SUBAPPLICATION HebenSenken_ILOCK_QDA_PWM_OPC (* 2 Remote-Kommandos (Heben/Senken, je Subscribe+State-Publish, ODER-verknuepft mit IO-Test wie bei ILOCK_SWITCH_2_QXA_OPC) auf 1 ratiometrisches PWM-Signal (Danfoss PVEA: 25%=Senken, 50%=Neutral, 75%=Heben, Lastteiler-korrigiert). ILOCK_SWITCH_PROTECT_AX (Last-Wins mit Schutzzeit) sorgt dafuer, dass Heben und Senken nie gleichzeitig aktiv sind. Generisch fuer jeden PVEA-Aktor mit ratiometrischem 3-Stufen-PWM-Kanal. *)
  (* Standard: 61499-2 *)
  (* Version 1.3, 2026-09-27, Franz Höpfinger, Meisterschulen am Ostbahnhof, Franz: 'HebenSenken_ILOCK_QDA_PWM_OPC sehe ich KEINE Aenderung?' - das eigene Mux/Skalierungs/Ausgabe-Teilnetz (ASSEMBLE_AB_FROM_AX/AB_TO_AUI/values_50_75_25/AR_AUI_MUX_3/AR_R_MUL_Korrektur/AR_R_MUL_PWM13BIT/AR_TO_AD_NUM/DigitalOutput_PWM) war seit der Auslagerung nach MyLib::sys::HebenSenken_QDA_PWM (fuer Bunkerboden_PWM) doppelt vorhanden - jetzt durch eine Instanz von HebenSenken_QDA_PWM ersetzt (HEBEN/SENKEN aus SPLIT_HEBEN_OUT/SPLIT_SENKEN_OUT direkt verdrahtet statt vorher inline), unveraendertes Verhalten, keine Duplizierung mehr. *)
  (* Version 1.2, 2026-09-27, Franz Höpfinger, Meisterschulen am Ostbahnhof, AR_R_MUL_Korrektur/AR_R_MUL_PWM13BIT FACTOR von eingebackenen Rohwerten (REAL#0.715/REAL#81.91) auf benannte Konstanten aus der neuen MyLib::sys::const::PWM_Konstanten umgestellt (PWM_LASTTEILER_KORREKTUR/PWM_13BIT_SKALIERUNG) - unveraendertes Verhalten, nur nicht mehr an mehreren Stellen als Rohwert wiederholt. values_50_75_25 bekommt jetzt explizit FACTOR_75/FACTOR_25 aus derselben GCF (VALUES_50_75_25_FACTOR_75/_25), seit values_50_75_25 v1.2 eigene Parameter statt eingebackener Werte. *)
  (* Version 1.1, 2026-09-20, Franz Höpfinger, Meisterschulen am Ostbahnhof, PWM_POW von intern fest verdrahtetem initval_AR (1.0) auf einen eigenen Socket umgestellt - ein generischer, wiederverwendbarer Typ darf keinen Fixwert fuer eine Groesse verdrahten, die pro Instanz unterschiedlich sein soll (z.B. Aufnahme_Rechts_KVE16_Reserve.SUB braucht ggf. eine andere Verdrahtung als Aufnahme_Links). *)
  (* Version 1.0, 2026-09-08, Franz Höpfinger, Meisterschulen am Ostbahnhof, Ausgelagert aus Heben_Senken_TO_QDA_PWM_OPC (PWM/ILOCK/Mux-Teilnetz, ohne die Freigabe-DO) zur Wiederverwendung. *)
  PACKAGE MyLib::sys;
  IMPORT logiBUS::io::DQ::logiBUS_DO;
  IMPORT logiBUS::io::DQ::logiBUS_DO_S;
  IMPORT MyLib::sys::const::PWM_Konstanten::PWM_LASTTEILER_KORREKTUR;
  IMPORT MyLib::sys::const::PWM_Konstanten::PWM_13BIT_SKALIERUNG;
  IMPORT MyLib::sys::const::PWM_Konstanten::VALUES_50_75_25_FACTOR_75;
  IMPORT MyLib::sys::const::PWM_Konstanten::VALUES_50_75_25_FACTOR_25;
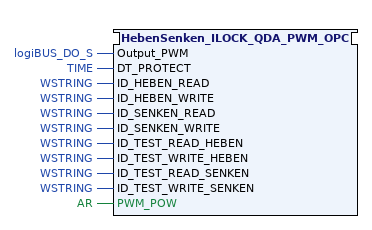
  VAR_INPUT
    Output_PWM : logiBUS::io::DQ::logiBUS_DO_S := logiBUS_DO::Invalid; (* Physischer PWM-Ausgang: 25/50/75% Tastgrad, ratiometrisch *)
    DT_PROTECT : TIME := T#300ms; (* Schutz-Totzeit vor Richtungswechsel *)
    ID_HEBEN_READ : WSTRING; (* Echtes Funktions-Kommando Heben (Subscribe) *)
    ID_HEBEN_WRITE : WSTRING; (* Echte Funktions-Rueckmeldung Heben, HINTER dem ILOCK (Publish) *)
    ID_SENKEN_READ : WSTRING; (* Echtes Funktions-Kommando Senken (Subscribe) *)
    ID_SENKEN_WRITE : WSTRING; (* Echte Funktions-Rueckmeldung Senken, HINTER dem ILOCK (Publish) *)
    ID_TEST_READ_HEBEN : WSTRING; (* Bestehende IO-Test-Subscribe-Adresse Heben (z.B. STG2_Q0x_READ), ODER-verknuepft mit ID_HEBEN_READ vor dem ILOCK *)
    ID_TEST_WRITE_HEBEN : WSTRING; (* Bestehende IO-Test-Publish-Adresse Heben, HINTER dem ILOCK (z.B. STG2_Q0x_WRITE) *)
    ID_TEST_READ_SENKEN : WSTRING; (* Bestehende IO-Test-Subscribe-Adresse Senken, ODER-verknuepft mit ID_SENKEN_READ vor dem ILOCK *)
    ID_TEST_WRITE_SENKEN : WSTRING; (* Bestehende IO-Test-Publish-Adresse Senken, HINTER dem ILOCK *)
  END_VAR
  SOCKETS
    PWM_POW : adapter::types::unidirectional::AR; (* PWM Power 1.0 = Maximale Power, 0.0 = Aus, 0.5 = Halb - durchgereicht an values_50_75_25.PWM_POW *)
  END_SOCKETS
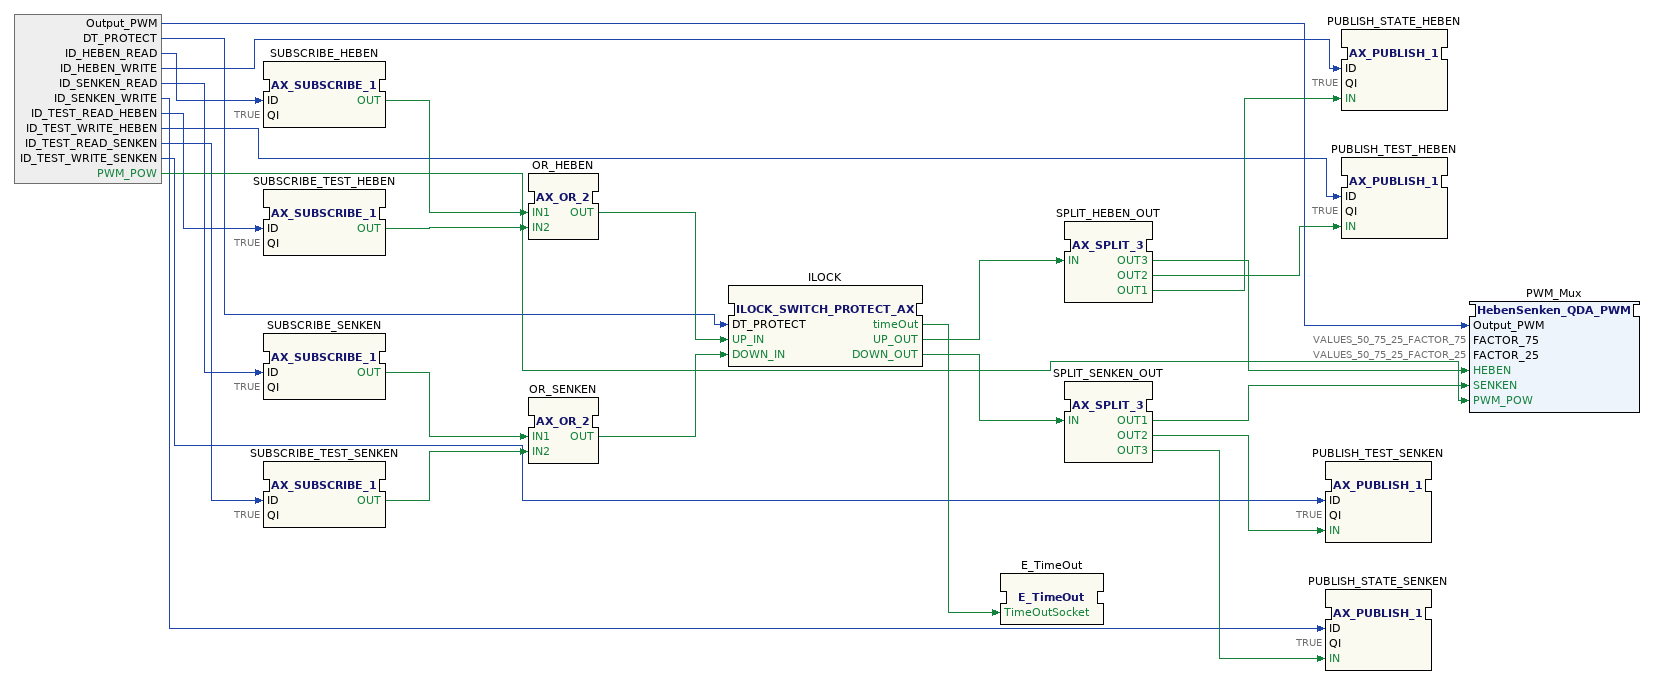
  FBS
    SUBSCRIBE_HEBEN : adapter::net::AX_SUBSCRIBE_1(QI := TRUE);
    SUBSCRIBE_TEST_HEBEN : adapter::net::AX_SUBSCRIBE_1(QI := TRUE);
    OR_HEBEN : adapter::booleanOperators::AX_OR_2;
    SUBSCRIBE_SENKEN : adapter::net::AX_SUBSCRIBE_1(QI := TRUE);
    SUBSCRIBE_TEST_SENKEN : adapter::net::AX_SUBSCRIBE_1(QI := TRUE);
    OR_SENKEN : adapter::booleanOperators::AX_OR_2;
    ILOCK : logiBUS::signalprocessing::interlock::ILOCK_SWITCH_PROTECT_AX;
    E_TimeOut : iec61499::events::E_TimeOut;
    SPLIT_HEBEN_OUT : adapter::events::unidirectional::AX_SPLIT_3;
    SPLIT_SENKEN_OUT : adapter::events::unidirectional::AX_SPLIT_3;
    PUBLISH_TEST_HEBEN : adapter::net::AX_PUBLISH_1(QI := TRUE);
    PUBLISH_STATE_HEBEN : adapter::net::AX_PUBLISH_1(QI := TRUE);
    PUBLISH_TEST_SENKEN : adapter::net::AX_PUBLISH_1(QI := TRUE);
    PUBLISH_STATE_SENKEN : adapter::net::AX_PUBLISH_1(QI := TRUE);
  END_FBS
  SUBAPPS
    PWM_Mux : MyLib::sys::HebenSenken_QDA_PWM(FACTOR_75 := VALUES_50_75_25_FACTOR_75, FACTOR_25 := VALUES_50_75_25_FACTOR_25); (* Mux/Skalierungs/Ausgabe-Teil (ASSEMBLE_AB_FROM_AX/AB_TO_AUI/values_50_75_25/AR_AUI_MUX_3/AR_R_MUL_Korrektur/AR_R_MUL_PWM13BIT/AR_TO_AD_NUM/DigitalOutput_PWM) ausgelagert - ILOCK_SWITCH_PROTECT_AX (Last-Wins mit Schutzzeit DT_PROTECT) sorgt weiterhin dafuer, dass HEBEN/SENKEN nie gleichzeitig aktiv sind. *)
  END_SUBAPPS
  DATA_CONNECTIONS
    ID_HEBEN_READ TO SUBSCRIBE_HEBEN.ID;
    ID_TEST_READ_HEBEN TO SUBSCRIBE_TEST_HEBEN.ID;
    ID_TEST_WRITE_HEBEN TO PUBLISH_TEST_HEBEN.ID;
    ID_HEBEN_WRITE TO PUBLISH_STATE_HEBEN.ID;
    ID_SENKEN_READ TO SUBSCRIBE_SENKEN.ID;
    ID_TEST_READ_SENKEN TO SUBSCRIBE_TEST_SENKEN.ID;
    ID_TEST_WRITE_SENKEN TO PUBLISH_TEST_SENKEN.ID;
    ID_SENKEN_WRITE TO PUBLISH_STATE_SENKEN.ID;
    Output_PWM TO PWM_Mux.Output_PWM;
    DT_PROTECT TO ILOCK.DT_PROTECT;
  END_CONNECTIONS
  ADAPTER_CONNECTIONS
    SUBSCRIBE_HEBEN.OUT TO OR_HEBEN.IN1;
    SUBSCRIBE_TEST_HEBEN.OUT TO OR_HEBEN.IN2;
    OR_HEBEN.OUT TO ILOCK.UP_IN;
    SUBSCRIBE_SENKEN.OUT TO OR_SENKEN.IN1;
    SUBSCRIBE_TEST_SENKEN.OUT TO OR_SENKEN.IN2;
    OR_SENKEN.OUT TO ILOCK.DOWN_IN;
    ILOCK.timeOut TO E_TimeOut.TimeOutSocket;
    ILOCK.UP_OUT TO SPLIT_HEBEN_OUT.IN;
    SPLIT_HEBEN_OUT.OUT3 TO PWM_Mux.HEBEN;
    SPLIT_HEBEN_OUT.OUT2 TO PUBLISH_TEST_HEBEN.IN;
    ILOCK.DOWN_OUT TO SPLIT_SENKEN_OUT.IN;
    SPLIT_SENKEN_OUT.OUT1 TO PWM_Mux.SENKEN;
    SPLIT_SENKEN_OUT.OUT2 TO PUBLISH_TEST_SENKEN.IN;
    SPLIT_SENKEN_OUT.OUT3 TO PUBLISH_STATE_SENKEN.IN;
    SPLIT_HEBEN_OUT.OUT1 TO PUBLISH_STATE_HEBEN.IN;
    PWM_POW TO PWM_Mux.PWM_POW;
  END_CONNECTIONS
END_SUBAPPLICATION
